// TIA Portal V17 export
// export: Created 2024-09-02T12:50:36.0879241Z, ExportSetting WithDefaults, DisplayName Totally Integrated Automation Portal, DisplayVersion V17, DisplayName TIA Portal Openness, DisplayVersion V17, DisplayName TIA Portal Version Control Interface, DisplayVersion V17, DisplayName STEP 7 Professional, DisplayVersion V17, DisplayName STEP 7 Safety, DisplayVersion V17, DisplayName WinCC Professional, DisplayVersion V17
TYPE "TypeMobyDMC_1"
// stored: IsFailsafeCompliant false
   STRUCT
      ZEICHEN : Array[1..64] of Char;
   END_STRUCT;
END_TYPE
